Universal Robots URScript: claude_trajectory_safe_move_j.script

# claude_trajectory_safe_move_j
#
# New template. A blended joint-interpolated trajectory with a force guard - the
# force-monitored equivalent of claude_trajectory_unsafe_move_j.script.
#
# There was no guarded trajectory template at all: safe_move_j / safe_move_l
# guard a single move, and the moment a motion is expressed as a waypoint list it
# silently loses its force guard. A blended path is exactly the case where a
# guard matters most, because it is the long unattended motion.
#
# The waypoint progress the guard reports is what makes a force stop recoverable:
# socket_server counts the waypoints that were reached, and
# handle_request::remaining_command drops those from the command so a resume
# continues forward instead of replaying the path from the start.
#
# force_threshold <= 0.0 disables the guard, matching claude_safe_move_*.
# Optional parameters: use_zero_ftsensor (true), force_settle_time (0.3),
# stop_acceleration (5.0).
#   check_safety_limits (true) - also check the target against the active safety
#                                planes, joint limits and tool orientation limit,
#                                not only whether inverse kinematics has a
#                                solution. This is what catches a pose that is
#                                reachable but would trip a protective stop.

global cl_move_done = False
global cl_force_detected = False
global cl_threshold = 0.0
global cl_settle = 0.0
global cl_base_f = [0.0, 0.0, 0.0, 0.0, 0.0, 0.0]
global cl_peak = 0.0
global cl_v = 0.0
global cl_a = 0.0

def script():
  cl_move_done = False
  cl_force_detected = False
  cl_peak = 0.0
  cl_threshold = {{ force_threshold }}
  cl_settle = {{ force_settle_time | default(value=0.3) }}

  {%- if use_payload %}
  set_target_payload({{ payload }})
  {%- endif %}
  set_tcp({{ tcp_in_faceplate }})

  {%- if waypoints | length == 0 %}
  socket_send_line("This is a trajectory command but no waypoints were given.", "ur_driver_socket")
  return False
  {%- endif %}

  socket_send_line("Validating guarded trajectory of {{ waypoints | length }} waypoints...", "ur_driver_socket")

  # --- PHASE 1: everything that can be checked without moving ---
  {%- for wp in waypoints %}
  {%- if not wp.use_joint_positions %}
  if point_dist({{ wp.target_in_base }}, p[0.0, 0.0, 0.0, 0.0, 0.0, 0.0]) < 0.001:
    socket_send_line("Waypoint {{ loop.index0 }} has an unset target (base origin). Refusing to move there.", "ur_driver_socket")
    return False
  end
  if not get_inverse_kin_has_solution({{ wp.target_in_base }}
    {%- if wp.use_preferred_joint_config -%}
    , qnear={{ wp.preferred_joint_config }}
    {%- endif -%}):
    socket_send_line("No inverse kinematics solution for waypoint {{ loop.index0 }}, aborting.", "ur_driver_socket")
    return False
  end
  {%- if check_safety_limits | default(value=true) %}
  if not is_within_safety_limits({{ wp.target_in_base }}):
    socket_send_line("Waypoint {{ loop.index0 }} is outside the active safety limits, aborting.", "ur_driver_socket")
    return False
  end
  {%- endif %}
  {%- endif %}
  {%- endfor %}

  if cl_threshold > 0.0:
    {%- if use_zero_ftsensor | default(value=true) %}
    zero_ftsensor()
    {%- endif %}
    sleep(0.1)
    cl_base_f = get_tcp_force()
  else:
    socket_send_line("force_threshold is 0, force monitoring is disabled for this trajectory.", "ur_driver_socket")
  end

  socket_send_line("Validation passed. Starting guarded continuous motion.", "ur_driver_socket")

  thread move_thread():
    {%- for wp in waypoints %}
    cl_v = {{ wp.velocity }}
    cl_a = {{ wp.acceleration }}
    if {{ wp.global_velocity_scaling }} > 0.0 and {{ wp.global_velocity_scaling }} <= 1.0:
      cl_v = cl_v * {{ wp.global_velocity_scaling }}
    end
    if {{ wp.global_acceleration_scaling }} > 0.0 and {{ wp.global_acceleration_scaling }} <= 1.0:
      cl_a = cl_a * {{ wp.global_acceleration_scaling }}
    end
    {%- if wp.use_joint_positions %}
    movej({{ wp.joint_positions }}, a=cl_a, v=cl_v
    {%- if wp.use_execution_time -%}
    , t={{ wp.execution_time }}
    {%- endif -%}
    {%- if wp.use_blend_radius -%}
    , r={{ wp.blend_radius }}
    {%- endif -%})
    {%- else %}
    movej({{ wp.target_in_base }}, a=cl_a, v=cl_v
    {%- if wp.use_execution_time -%}
    , t={{ wp.execution_time }}
    {%- endif -%}
    {%- if wp.use_blend_radius -%}
    , r={{ wp.blend_radius }}
    {%- endif -%})
    {%- endif %}
    {%- endfor %}
    cl_move_done = True
  end

  thread force_monitor_thread():
    if cl_threshold > 0.0:
      sleep(cl_settle)
      while not cl_move_done:
        w = get_tcp_force()
        dx = w[0] - cl_base_f[0]
        dy = w[1] - cl_base_f[1]
        dz = w[2] - cl_base_f[2]
        mag = sqrt(dx * dx + dy * dy + dz * dz)
        if mag > cl_peak:
          cl_peak = mag
        end
        if mag > cl_threshold:
          cl_force_detected = True
          break
        end
        sleep(0.002)
      end
    end
  end

  {%- if report_waypoint_progress %}
  thread progress_thread():
    {%- for wp in waypoints %}
    {%- if wp.use_joint_positions %}
    while point_dist(get_actual_tcp_pose(), get_forward_kin({{ wp.joint_positions }})) > {% if wp.use_blend_radius %}{{ wp.blend_radius * 1.5 + 0.005 | round(precision=4) }}{% else %}0.005{% endif %}:
      sleep(0.004)
    end
    {%- else %}
    while point_dist(get_actual_tcp_pose(), {{ wp.target_in_base }}) > {% if wp.use_blend_radius %}{{ wp.blend_radius * 1.5 + 0.005 | round(precision=4) }}{% else %}0.005{% endif %}:
      sleep(0.004)
    end
    {%- endif %}
    socket_send_line("waypoint_reached {{ loop.index0 }}", "ur_driver_socket")
    {%- endfor %}
  end
  t_progress = run progress_thread()
  {%- endif %}

  t_move = run move_thread()
  t_force = run force_monitor_thread()

  while not cl_move_done and not cl_force_detected:
    sleep(0.002)
  end

  {%- if report_waypoint_progress %}
  sleep(0.05)
  kill t_progress
  {%- endif %}
  kill t_move
  kill t_force
  stopj({{ stop_acceleration | default(value=5.0) }})
  sleep(0.5)

  if cl_force_detected:
    socket_send_line("force_stop peak=" + to_str(cl_peak) + "N threshold=" + to_str(cl_threshold) + "N", "ur_driver_socket")
    return False
  end
  return cl_move_done
end
